FUNCTION_BLOCK FB_1_SituarBase_SFC
VAR_INPUT
	
	//  SFC-Flags
	SFCPause: BOOL;
	SFCReset: BOOL;

	// Indicadores de sincronización
	Ack: BOOL := TRUE;
	Execute: BOOL;
	
	// Entradas
	PalePresencia: BOOL;
	TpoCintaDelSensorAlTope: TIME;
	
END_VAR
VAR_OUTPUT
	
	// Indicadores de sincronización
	Ready: BOOL;	
	Done: BOOL;
	
	// Salidas
	CintaMotorActiva: BOOL;
	
END_VAR
VAR
END_VAR

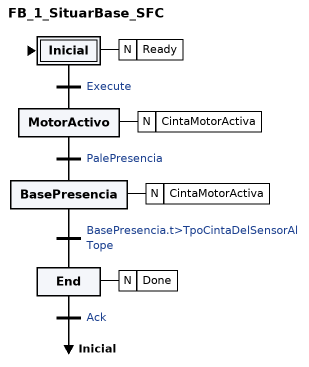
INITIAL_STEP Inicial:
    Ready(N);
END_STEP
TRANSITION FROM Inicial TO MotorActivo
    := Execute;
END_TRANSITION
STEP MotorActivo:
    CintaMotorActiva(N);
END_STEP
TRANSITION FROM MotorActivo TO BasePresencia
    := PalePresencia;
END_TRANSITION
STEP BasePresencia:
    CintaMotorActiva(N);
END_STEP
TRANSITION FROM BasePresencia TO End
    := BasePresencia.t>TpoCintaDelSensorAlTope;
END_TRANSITION
STEP End:
    Done(N);
END_STEP
TRANSITION FROM End TO Inicial
    := Ack;
END_TRANSITION

END_FUNCTION_BLOCK

(* stored: Version 1.1.0.1, ProductVersion 3.1.4024.12
   POU FB_1_SituarBase_SFC: Id {276a140a-178d-422b-a4dd-c4a88a49affb}, SpecialFunc None *)
